FUNCTION_BLOCK Real_Half (* Basic FB with empty ECC *)
  (* Standard: 61499-2; Description: Multiply real input with a half. *)
  (* Version 1.0, 2020-08-17, Candra Wardaya, UGM *)
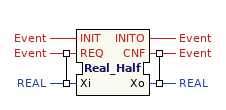
  EVENT_INPUT
    INIT; (* Initialization *)
    REQ WITH Xi; (* Execution Request *)
  END_EVENT
  EVENT_OUTPUT
    INITO; (* Output Initialization *)
    CNF WITH Xo; (* Confirmation of Execution *)
  END_EVENT
  VAR_INPUT
    Xi : REAL; (* Real Input *)
  END_VAR
  VAR_OUTPUT
    Xo : REAL; (* Real Output *)
  END_VAR
  VAR
    X : REAL; (* Internal Variable *)
  END_VAR
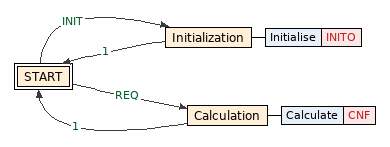
  EC_STATES
    START; (* Initial State *)
    Initialization : Initialise -> INITO;
    Calculation : Calculate -> CNF;
  END_STATES
  EC_TRANSITIONS
    START TO Initialization := INIT;
    Initialization TO START := 1;
    START TO Calculation := REQ;
    Calculation TO START := 1;
  END_TRANSITIONS
  ALGORITHM Initialise IN ST: (* New Algorithm *)

  END_ALGORITHM
  ALGORITHM Calculate IN ST: (* New Algorithm *)
Xo := Xi*0.5;
  END_ALGORITHM
END_FUNCTION_BLOCK
